# EPICS SNL sequencer program: VCSIOCS/cnAIOC/cnAiocApp/src/cnaClearanceSNC.stt
program cnaClearanceSNC

%{
#include "vcs_var_mes.h" // define this here so C functions are seen
#define STOK        0
#define WFVC        55
#define	B39OFF      122
#define	B38ON       121
#define DA12AS1OFF   123
#define DA12AS2OFF   124
#define cnAPNK      119
}%

/* Declare seq variables*/
/* Declare seq variables*/
short cnA_INIT;
short cnA_VC;
short cnA_W38_STS;
short cnA_W39_STS;
short cnA_FAIL_COND;
short cnA_PNK;
short cnA_RST_OUTS;
string cnA_CLR_STATS;
string cnA_INTLCK_STATS;
// CONTROL FLAGS
short cnA_failed_rst;
short cnA_OLD_FAIL_COND;
short cnA_not_cleared = FALSE;

/* Associate SNL variables with epics output pv's*/
assign	cnA_RST_OUTS        to	"{SYS}:RST-cnA.PROC";
assign	cnA_CLR_STATS       to	"{SYS}:cnA-CLR-STATS";
assign	cnA_INTLCK_STATS	to  "{SYS}:cnA-INTLCK-STATS";

/* Associate SNL variables with epics input pv's*/
assign 	cnA_VC 		        to 	"{SYS}:cnA-VC";
assign 	cnA_W38_STS 		to 	"{SYS}:cnA-W38-STS";
assign 	cnA_W39_STS 		to 	"{SYS}:cnA-W39-STS";
assign	cnA_FAIL_COND		to  "{SYS}:cnA-FAIL-COND";
assign	cnA_PNK		        to  "{SYS}:cnA-PNK";

monitor	cnA_VC;
monitor cnA_W38_STS;
monitor cnA_W39_STS;
monitor	cnA_FAIL_COND;
monitor	cnA_PNK;

ss cnA_clearance_status {

    state init {
		  when (delay(1)) {
			  initVault();
			  printf("\n%scnA VAULT INITIALISATION COMPLETED%s\n",OK,DEF);
		  }   state watchman_38_pressed
    }
//////////////////////////////////////////////////////////
	state watchman_38_pressed {

    when (cnA_FAIL_COND != STOK) {
      cnA_OLD_FAIL_COND = cnA_FAIL_COND;
    } state  clearance_faillures

		when (cnA_W38_STS == WFVC) {

		} state clearance_pending

		when (cnA_W38_STS == B38ON) {
			cnA_clear_underway();
			cnA_update_report(B38ON);
		} state watchman_38_released
	}
 ////////////////////////////////////////////////////////////////
	state clearance_pending {
		option -e;
		option -x;
		entry {
      resetVault();
      cnA_update_report(WFVC);
      cnA_not_cleared = TRUE; // we use this to tell user to start or restart vault clearance
		}
		when (cnA_W38_STS != WFVC) {

		} state watchman_38_pressed
	}
 //////////////////////////////////////////////////////////
	state watchman_38_released {

		when (cnA_FAIL_COND != STOK) {

		} state  clearance_faillures

		when (cnA_W38_STS != B38ON) {

		} state A12A_switch_I_closed
	}
//////////////////////////////////////////////////////////
	state A12A_switch_I_closed {

		option -e;

		entry {
      cnA_update_report(DA12AS1OFF);
		}

		when (cnA_FAIL_COND != STOK) {

		} state   clearance_faillures

		when (cnA_W39_STS != DA12AS1OFF) {

		} state A12A_switch_II_closed

	}
 //////////////////////////////////////////////////////////
	state A12A_switch_II_closed {

		option -e;

		entry {
      cnA_update_report(DA12AS2OFF);
		}

		when (cnA_FAIL_COND != STOK) {

		} state   clearance_faillures

   // previous switch might have opened up
		when (cnA_W39_STS == DA12AS1OFF) {

		} state A12A_switch_I_closed

		when (cnA_W39_STS != DA12AS2OFF) {

		} state watchman_39_pressed
	}
///////////////////////////////////////////////////////////
	state watchman_39_pressed {

		option -e;

		entry {
      cnA_update_report(B39OFF);
		}

		when (cnA_FAIL_COND != STOK) {

		} state  clearance_faillures

		when (cnA_W39_STS == STOK) {
		} state vault_cleared

   /// must be last
		when (cnA_W39_STS != B39OFF) {

		} state A12A_switch_I_closed
	}
///////////////////////////////////////////////////////////////
  state vault_cleared {
		option -e;
		entry {
      cnA_status();
			printf("%scnA VAULT IN CLEARED STATE%s\n",CLR,DEF);
		}
		when (cnA_VC != STOK) {

		} state paniq_faillure

	}
 ///////////////////////////////////////////////////
  state paniq_faillure {

    when (cnA_VC != cnAPNK) {

		} state clearance_faillures

    when () { // paniq button released?
      printf("cnA VAULT CLEARED FAILURE CONDITION: ");
      cnA_update_failed(cnAPNK);
		} state recover_from_paniq
	}
////////////////////////////////////////////////////////////
  state recover_from_paniq {
		option -e;
		option -x;
		when (!cnA_PNK) { // paniq button released?
        // we only go to this state so we enter watchman_38_pressed from one point(recover_from_faillure)
		} state recover_from_faillure

		exit {
      cnA_failed_rst = FALSE;
      cnA_not_cleared = FALSE;
      //printf("%scnA RECOVERING FROM PANIQ FAILLURE : ENTERING W38 STATE%s\n",OK,DEF);
		}
	}
 ///////////////////////////////////////////////////
  state clearance_faillures {
		option -e;
		option -x;
		entry {
            printf("cnA CLEARANCE FAILURE CONDITION: ");
            cnA_failed_rst = FALSE;
            cnA_not_cleared = FALSE;
            cnA_OLD_FAIL_COND = cnA_FAIL_COND;
            cnA_update_failed(cnA_FAIL_COND); // we cannot index -1(FAIL)
		}

		when () { // seq excute faster than recor logi
		} state recover_from_faillure
	}
//////////////////////////////////////////////////////////
	state recover_from_faillure {

		when (cnA_FAIL_COND ==  STOK) {
      printf("%scnA RECOVERING FROM CLEARANCE  FAILLURE : ENTERING W38 STATE%s\n",OK,DEF);
		} state  watchman_38_pressed

		when (cnA_FAIL_COND != cnA_OLD_FAIL_COND) {

		} state  clearance_faillures
	}
}
///////////////////////////////////////////////////////////////////////////////
void initVault(){
  cnA_OLD_FAIL_COND = cnA_FAIL_COND;
  cnA_RST_OUTS  = TRUE;
	not_cleared(cnA_CLR_STATS);
	report_error(cnA_INTLCK_STATS, 0);
  pvPut(cnA_RST_OUTS, SYNC);
	pvPut(cnA_CLR_STATS, SYNC);
	pvPut(cnA_INTLCK_STATS, SYNC);
}
////////////////////////////////////////////////////////////////////////
void resetVault(){
	not_cleared(cnA_CLR_STATS);
	pvPut(cnA_CLR_STATS, SYNC);
}
////////////////////////////////////////////////////////////////////////
void cnA_update_failed(short report)
{
	clear_failed(cnA_CLR_STATS);
	pvPut(cnA_CLR_STATS, SYNC);
	report_error(cnA_INTLCK_STATS, report);
	pvPut(cnA_INTLCK_STATS, SYNC);
	printf("%s%s%s\n",ERROR,cnA_INTLCK_STATS,DEF);
}
/////////////////////////////////////////////////////////////////////////
void cnA_update_report(short intlck) {
	report_error(cnA_INTLCK_STATS, intlck);
	pvPut(cnA_INTLCK_STATS, SYNC);
}
////////////////////////////////////////////////////////////////////////
void cnA_status()
{
	cleared(cnA_CLR_STATS);
	pvPut(cnA_CLR_STATS, SYNC);
	report_error(cnA_INTLCK_STATS, 0);
	pvPut(cnA_INTLCK_STATS, SYNC);
}
///////////////////////////////////////////////////////////
void cnA_clear_underway()
{
	clear_underway(cnA_CLR_STATS);
	pvPut(cnA_CLR_STATS, SYNC);
}

//////////////////////////////////////////////////////////////////////////
%{

inline void cleared(string vault_status) {
    strcpy(vault_status, mes_array[1]); // Area cleared
}
////////////////////////////////////////////////
inline void not_cleared(string vault_status) {
   strcpy(vault_status, mes_array[2]); // Area not cleared
}
///////////////////////////////////////////////
inline void clear_underway(string vault_status) {
   strcpy(vault_status, mes_array[3]);  // Area clearance underway
}
//////////////////////////////////////////////
inline void clear_failed(string vault_status) {
   strcpy(vault_status, mes_array[5]); // Area clearance fail
}
////////////////////////////////////////////////
inline void report_error(string vault_interlock, short intlock)
{
   strcpy(vault_interlock, mes_array[intlock]);
}

}%
